Yaskawa INFORM job: BATMAN_4SPOINY2.JBI

/JOB
//NAME BATMAN_4SPOINY2
///FOLDERNAME KRIS-SCIANA
//POS
///NPOS 293,293,292,19,0,0
///TOOL 0
///POSTYPE PULSE
///PULSE
C00000=-27461,19727,-15013,-5964,93200,-7919
C00001=-53930,-34836,-43070,-10546,92631,44102
C00002=-59372,-32233,-36195,-10185,89087,42536
C00003=-59542,-32241,-35992,-10174,88938,42491
C00004=-59542,-32044,-34623,-10174,88208,42551
C00005=-59542,-32113,-35077,-10174,88448,42531
C00006=-60552,-31800,-34867,-10107,88354,42193
C00007=-59542,-32241,-35992,-10174,88938,42491
C00008=-64039,-48991,-58660,-9906,93649,40580
C00009=-69362,-49546,-56329,-9460,91325,38954
C00010=-72521,-45533,-52121,-9188,90441,37947
C00011=-72521,-45462,-50975,-9185,89780,37995
C00012=-72775,-45521,-51067,-9161,89777,37907
C00013=-73792,-45251,-50904,-9073,89701,37568
C00014=-72521,-45533,-52121,-9188,90441,37947
C00015=-72780,-67210,-74355,-9190,92926,37677
C00016=-104760,-79002,-75488,-1590,83769,-10908
C00017=-104760,-78316,-71792,-1595,81848,-10885
C00018=-104951,-72146,-66630,-1566,81838,-10949
C00019=-104951,-71873,-65349,-1567,81190,-10942
C00020=-104951,-71915,-65543,-1567,81288,-10943
C00021=-104860,-69153,-64201,-1578,81883,-10919
C00022=-104951,-72146,-66630,-1566,81838,-10949
C00023=-126930,-89810,-77004,2546,79326,-20912
C00024=-126930,-86182,-66696,2587,74851,-21005
C00025=-124517,-79688,-62407,2239,75475,-20152
C00026=-124517,-79051,-60693,2247,74749,-20166
C00027=-124517,-79260,-61250,2244,74984,-20162
C00028=-123686,-77088,-60280,2122,75480,-19864
C00029=-124517,-79688,-62407,2239,75475,-20152
C00030=-203387,-120314,-87249,1260,66339,-1853
C00031=-200667,-112422,-82916,708,67693,-857
C00032=-200667,-111236,-80756,708,66973,-859
C00033=-200667,-111296,-80865,708,67010,-859
C00034=-200121,-107908,-79763,595,68068,-656
C00035=-200667,-112422,-82916,708,67693,-857
C00036=-197903,-118206,-84689,161,65798,138
C00037=-190700,-136110,-79236,-12987,43309,5470
C00038=-193247,-133524,-78729,-11658,43940,4204
C00039=-193037,-133750,-78775,-11768,43882,4308
C00040=-191788,-131166,-76340,-12346,43888,4881
C00041=-190700,-136110,-79236,-12987,43309,5470
C00042=-159264,-85348,-72338,-26469,101848,35770
C00043=-164489,-85917,-58916,-26689,92487,35917
C00044=-168795,-82306,-57912,-27368,92208,34361
C00045=-170153,-80945,-57335,-27563,92069,33880
C00046=-170038,-81063,-57386,-27546,92081,33921
C00047=-169577,-79396,-55147,-27467,91768,34169
C00048=-168310,-82776,-58110,-27297,92259,34533
C00049=-174818,-166728,-104111,-5010,53468,9061
C00050=-151913,-165072,-108467,-9162,58894,17426
C00051=-31054,-58499,-67437,4813,86361,-7552
C00052=-17460,-13489,-32841,-5083,88285,10080
C00053=-18511,-10450,-28211,-4896,86939,9785
C00054=-18511,-10517,-26393,-4896,85789,9828
C00055=-18511,-10513,-26589,-4896,85911,9823
C00056=-19077,-8695,-25164,-4796,85935,9632
C00057=-18511,-10450,-28211,-4896,86939,9785
C00058=-19304,-17015,-37138,-4755,89006,9443
C00059=-40718,-16031,-27821,22618,89289,-5458
C00060=-35897,-12993,-23126,22071,86757,-4185
C00061=-35281,-10295,-21039,21995,86689,-3974
C00062=-35332,-10522,-21216,22001,86695,-3991
C00063=-35622,-10102,-19772,22045,86146,-4196
C00064=-35897,-12993,-23126,22071,86757,-4185
C00065=-31722,-22647,-27301,21597,83426,-3277
C00066=-29589,-18207,-23578,21312,82862,-2603
C00067=-29146,-15879,-21843,21245,82867,-2441
C00068=-29176,-16038,-21963,21249,82867,-2452
C00069=-29589,-15481,-20299,21334,82283,-2705
C00070=-29589,-18207,-23578,21312,82862,-2603
C00071=-33057,-35215,-50272,21725,90936,-2406
C00072=-13245,-10427,-29720,-5825,88219,11479
C00073=-13392,-4620,-21957,-5803,86422,11510
C00074=-18089,-7824,-24653,-4974,86126,9958
C00075=-18110,-8277,-24801,-4969,85982,9956
C00076=-21731,-10101,-26115,-4319,85651,8761
C00077=-21661,-10606,-26277,-4332,85495,8790
C00078=-25333,-12975,-27458,1213,84432,-1078
C00079=-19736,-16503,-27105,153,82354,789
C00080=-19363,-16615,-23205,6723,81452,-11372
C00081=-19940,-18075,-23614,6826,80998,-11595
C00082=-21964,-21673,-24603,7190,79942,-12350
C00083=-17410,-32379,-43825,-1943,88285,-427
C00084=-62758,-61083,-67514,-9356,96495,-3913
C00085=-199419,-126821,-93595,3849,72358,-1575
C00086=-214502,-101666,-82310,5387,79190,-6557
C00087=-215506,-95023,-76790,5488,79275,-6899
C00088=-206115,-95822,-76918,4502,78358,-3694
C00089=-205954,-96216,-76904,4488,78140,-3647
C00090=-199122,-96202,-76993,3725,77851,-1303
C00091=-199042,-96881,-76975,3719,77487,-1286
C00092=-188080,-119856,-79732,-8116,56883,3611
C00093=-198128,-125068,-78160,-5331,52444,-116
C00094=-199195,-125100,-74360,-11289,52271,7622
C00095=-182925,-108601,-69012,-21109,69501,28632
C00096=-173900,-101221,-64126,-22433,76310,30875
C00097=-171717,-100952,-63344,-22409,76572,31621
C00098=-165785,-126013,-84565,-21580,74443,34035
C00099=-65346,-79799,-84675,-10403,98195,30166
C00100=-73114,-35172,-46632,-9001,95792,24844
C00101=-73893,-33313,-43666,-8951,94846,24646
C00102=-56936,-3129,-12114,-26947,108321,27456
C00103=-55222,-19377,-25500,-26230,99599,30116
C00104=-48000,-22204,-22466,-25349,98847,33036
C00105=-47657,-23151,-32449,-25918,104076,32001
C00106=-58332,-49897,-67983,-12473,95404,30979
C00107=-76814,-87681,-77913,-12459,85852,4883
C00108=-98077,-64526,-65270,-10461,86864,-2540
C00109=-98077,-64172,-62734,-10473,85508,-2426
C00110=-98453,-62350,-60144,-10440,84814,-2496
C00111=-136928,-61997,-53571,24295,84631,-16368
C00112=-133428,-78274,-60683,19711,72960,-18904
C00113=-138454,-87211,-60543,20798,69473,-20912
C00114=-139028,-90281,-60991,20666,67739,-20449
C00115=-142002,-103150,-73880,19907,68072,-18980
C00116=-156669,-121711,-96887,11323,85539,-21769
C00117=-4467,-137969,-110669,6539,34039,3130
C00118=30106,49184,30056,7190,99242,80021
C00119=48667,-97469,-88024,4384,73291,-2494
C00120=49689,-78507,-72154,4117,73215,-2136
C00121=49303,-77230,-69865,4233,72483,-2298
C00122=49303,-77321,-70267,4229,72684,-2291
C00123=50594,-75678,-69509,3881,72996,-1827
C00124=50087,-79365,-72449,4017,72936,-2008
C00125=68843,-102719,-94603,-719,75306,4406
C00126=111940,-50312,-66287,845,90558,-21262
C00127=116747,-35795,-51410,28,88834,-19690
C00128=111075,-31135,-44901,14748,90637,-31106
C00129=112095,-31393,-44814,14616,90275,-30800
C00130=112020,-31375,-44802,14625,90290,-30824
C00131=111824,-29375,-42859,14647,90161,-30907
C00132=111075,-31135,-44901,14748,90637,-31106
C00133=115266,-12451,-41016,14369,96902,-28947
C00134=116842,-11754,-38964,14110,95764,-28553
C00135=117372,-11882,-38755,14027,95487,-28407
C00136=117096,-11854,-38735,14068,95534,-28493
C00137=116813,-10897,-37010,14093,95030,-28645
C00138=116549,-12463,-39204,14145,95601,-28669
C00139=116973,-27524,-54545,13255,91925,-29024
C00140=161629,-1767,-40127,-12706,111151,26907
C00141=160258,-5533,-27257,-16420,102000,26864
C00142=159800,-6307,-27168,-16383,101475,26773
C00143=160112,-5979,-26905,-16385,101541,26874
C00144=160141,-5574,-26041,-16363,101235,26926
C00145=160369,-6103,-29045,-16480,102795,26791
C00146=164567,12479,-21852,-12411,107740,28291
C00147=157312,-12873,-46942,3000,99665,-17174
C00148=206670,-20156,-47225,-4407,96533,-1302
C00149=207907,-5048,-28631,-4546,92932,-767
C00150=208193,-3786,-26509,-4582,92292,-649
C00151=208113,-4178,-26830,-4572,92282,-675
C00152=207509,-3531,-26303,-4488,92258,-873
C00153=208421,-5827,-28734,-4617,92624,-586
C00154=203791,-18365,-44572,-3987,95682,-2207
C00155=208102,-33244,-47535,-4348,72415,7516
C00156=208287,-28436,-43134,-4423,72190,7588
C00157=208434,-26310,-39925,-4502,71320,7672
C00158=208234,-36837,-41271,-4553,66735,7774
C00159=211009,-27621,-51707,-11614,93139,6311
C00160=152191,-52771,-83975,581,97487,43791
C00161=98829,-151569,-113617,-23423,60554,27083
C00162=63524,-95054,-80306,-9988,61383,12838
C00163=56536,-90563,-73566,-3171,58185,6546
C00164=56829,-88451,-72049,-3291,58345,6659
C00165=59876,-96663,-69219,-4945,52557,8119
C00166=60612,-96600,-68978,-5290,52489,8431
C00167=66960,-122601,-100767,717,65616,10335
C00168=151266,-17849,-52541,-13551,97671,36399
C00169=151622,-1723,-33362,-14991,96990,34005
C00170=151262,-1470,-31417,-14895,95899,34022
C00171=156478,-8848,-32076,-16260,93850,43651
C00172=161716,-19976,-35221,-16293,90376,44394
C00173=166380,-28542,-48041,-15538,92590,42053
C00174=176343,-26479,-59966,-14563,99290,38519
C00175=146432,-61605,-81283,-8581,90439,-5938
C00176=135076,-29257,-55178,-6049,90016,-9585
C00177=132700,-20433,-48103,-5503,90033,-10349
C00178=132491,-20005,-45954,-5452,88921,-10367
C00179=119630,-24773,-46451,11613,85271,-20135
C00180=112679,-48956,-51902,13552,77458,-23307
C00181=112569,-49156,-51831,13583,77335,-23359
C00182=106405,-53144,-61429,14838,82147,-24955
C00183=95224,-20248,-47255,12300,95289,-25611
C00184=95224,-20248,-47255,12300,95289,-25611
C00185=95567,-18089,-45671,12250,95373,-25491
C00186=-2669,-23033,-45877,12237,95351,-20479
C00187=-12882,-2605,-25335,12289,80797,-48712
C00188=-140228,6897,-12502,-16068,89102,25779
C00189=-178636,-27124,-21178,-9459,71149,14213
C00190=-190464,-2943,-638,1694,79970,9758
C00191=-190464,-2776,-23,1695,79677,9755
C00192=-190464,-2814,-164,1695,79744,9755
C00193=-190464,-1537,886,1697,79752,9755
C00194=-190079,-4348,-2686,1653,80502,9898
C00195=-170718,-9928,-4442,-11260,70728,17109
C00196=-176690,17572,15984,1100,84656,14555
C00197=-176690,17883,17124,1100,84116,14551
C00198=-176690,17847,16991,1100,84180,14551
C00199=-176937,19636,18668,1110,84073,14467
C00200=-176937,19636,18668,1110,84073,14467
C00201=-176690,17548,15886,1101,84706,14556
C00202=-159096,9684,11840,-13524,72569,21129
C00203=-163699,22746,22031,-3647,77400,19020
C00204=-163699,23053,23077,-3652,76914,19034
C00205=-163699,23004,22912,-3650,76991,19033
C00206=-164134,24645,24494,-3598,76842,18886
C00207=-163699,22706,21893,-3644,77465,19019
C00208=-150784,28408,29058,-15005,73089,24078
C00209=-157156,46221,45175,-1187,77129,21209
C00210=-157156,46539,46094,-1188,76728,21212
C00211=-157156,46464,45876,-1188,76822,21213
C00212=-157735,48153,47710,-1132,76554,21017
C00213=-157156,45966,44419,-1185,77462,21208
C00214=-142367,61055,63211,-16591,70629,27483
C00215=-154723,15756,14414,-2197,80088,22021
C00216=-154723,16062,15536,-2199,79553,22032
C00217=-154723,16000,15312,-2199,79658,22029
C00218=-155361,17628,16818,-2136,79550,21813
C00219=-154295,14517,12085,-2236,80891,22153
C00220=-151769,-34490,-30946,-14563,77368,23201
C00221=-173063,-38776,-28238,-10774,70233,16311
C00222=-172381,-31676,-18222,-12843,69119,19791
C00223=-189396,-43787,-25561,-9322,65102,13897
C00224=-212287,-48657,-28204,-3544,62394,5501
C00225=-221997,-47169,-27328,-892,62356,1858
C00226=-221072,-57002,-35060,1210,62084,-1011
C00227=-183831,-45924,-33017,621,66496,-211
C00228=-184325,-38707,-22706,764,63866,-409
C00229=-169590,-26315,-14874,-3175,65639,5020
C00230=-153390,-792,4257,-7245,68027,10841
C00231=-148403,11895,15303,-8450,68237,12643
C00232=-147332,15315,18416,-8713,68194,13036
C00233=-141966,-23744,-26450,-9578,76254,14345
C00234=-49773,-23801,-26487,-9571,76243,10777
C00235=-11499,-92934,-63711,-14704,67160,23123
C00236=5078,129767,24381,-2980,99042,84457
C00237=-23281,115763,31203,9131,91877,90037
C00238=-55336,37368,-13455,9130,92546,90074
C00239=-110497,-96700,-87975,9097,92672,90031
C00240=-122519,-98627,-88731,8985,93501,45120
C00241=-122519,-98627,-88731,8985,93501,45120
C00242=-231043,-103510,-90228,-14600,66848,14562
C00243=-239015,-52899,-63453,-12354,87389,13057
C00244=-232211,-37055,-48018,-13457,87263,15389
C00245=-232200,-37444,-47619,-13460,86829,15441
C00246=-232200,-37417,-46208,-13467,85999,15531
C00247=-232200,-37422,-46357,-13466,86086,15522
C00248=-232546,-36405,-45702,-13410,86146,15397
C00249=-232526,-38013,-47982,-13409,86709,15341
C00250=-213204,-18706,-38315,-16054,93998,21087
C00251=-215284,-13076,-30615,-15755,91824,20653
C00252=-215284,-13133,-29398,-15744,91072,20748
C00253=-215284,-13128,-29540,-15745,91159,20737
C00254=-215902,-11928,-28618,-15673,91088,20532
C00255=-215392,-13382,-30849,-15743,91789,20621
C00256=-206438,9841,-12512,-16716,94160,23395
C00257=-205120,11503,-10315,-16825,93948,23882
C00258=-205120,11440,-9133,-16804,93220,23984
C00259=-205120,11443,-9214,-16804,93269,23978
C00260=-205697,12454,-8305,-16750,93115,23798
C00261=-205222,11014,-10755,-16815,93943,23847
C00262=-210286,16144,-6103,-16310,92719,22261
C00263=-208996,19538,-3176,-16442,92919,22681
C00264=-208996,19485,-1978,-16424,92184,22779
C00265=-208996,19488,-2094,-16426,92254,22769
C00266=-209668,20896,-770,-16357,92032,22565
C00267=-208996,19564,-3616,-16449,93191,22643
C00268=-202176,43267,18401,-17042,93256,25006
C00269=-201249,45778,22861,-17085,92051,25496
C00270=-201249,45831,24224,-17069,91274,25603
C00271=-201249,45825,24100,-17070,91344,25593
C00272=-201817,46846,25195,-17022,91083,25430
C00273=-201596,44518,21658,-17057,92067,25371
C00274=-210187,6216,-22915,-16512,97781,21615
C00275=-216436,-2522,-24538,-15653,93231,20080
C00276=-219720,2451,-17856,-13270,92091,26137
C00277=-232169,-16488,-32780,-11683,89671,22159
C00278=-226973,-31382,-43065,-12371,89135,23971
C00279=-237194,-42183,-49809,-10971,86308,20756
C00280=-231421,-47421,-61288,-11801,91394,22246
C00281=-231421,-47421,-61288,-11801,91394,22246
C00282=-240248,-57151,-63303,-3936,83174,7432
C00283=-224450,-39830,-53255,-6930,86930,12556
C00284=-211441,-17782,-38439,-9211,90387,16662
C00285=-206434,-6086,-29592,-10033,91526,18242
C00286=-205798,-3820,-27691,-10133,91599,18448
C00287=-200228,-22351,-51424,-11111,97297,19798
C00288=-129551,-116321,-98683,-1361,90461,40912
C00289=-129551,-116321,-98683,-1361,90461,40912
C00290=-59952,-112124,-97380,-1385,91667,40557
C00291=-59953,-112125,-97379,-1385,91667,40556
C00292=1527,-36481,-34263,-1012,58134,86073
BC00000=81460,853554,487182
BC00001=164754,872951,482279
BC00002=164754,872951,482279
BC00003=164754,872951,482279
BC00004=164754,872951,482279
BC00005=164754,872951,482279
BC00006=164754,872951,482279
BC00007=164754,872951,482279
BC00008=164754,872951,482279
BC00009=164754,872951,482279
BC00010=164754,872951,482279
BC00011=164754,872951,482279
BC00012=164754,872951,482279
BC00013=164754,872951,482279
BC00014=164754,872951,482279
BC00015=164754,872951,482279
BC00016=164754,872951,482279
BC00017=164754,872951,482279
BC00018=164754,872951,482279
BC00019=164754,872951,482279
BC00020=164754,872951,482279
BC00021=164754,872951,482279
BC00022=164754,872951,482279
BC00023=164754,872951,482279
BC00024=164754,872951,482279
BC00025=164754,872951,482279
BC00026=164754,872951,482279
BC00027=164754,872951,482279
BC00028=164754,872951,482279
BC00029=164754,872951,482279
BC00030=164754,872951,482279
BC00031=164754,872951,482279
BC00032=164754,872951,482279
BC00033=164754,872951,482279
BC00034=164754,872951,482279
BC00035=164754,872951,482279
BC00036=164754,872951,482279
BC00037=164754,872951,482279
BC00038=164754,872951,482279
BC00039=164754,872951,482279
BC00040=164754,872951,482279
BC00041=164754,872951,482279
BC00042=164753,872951,482277
BC00043=164753,872950,482272
BC00044=164753,872950,482272
BC00045=164753,872950,482272
BC00046=164753,872950,482272
BC00047=164753,872950,482272
BC00048=164753,872950,482272
BC00049=164754,872951,482279
BC00050=164754,872951,482279
BC00051=164754,872951,482279
BC00052=164754,872951,482279
BC00053=164754,872951,482279
BC00054=164754,872951,482279
BC00055=164754,872951,482279
BC00056=164754,872951,482279
BC00057=164754,872951,482279
BC00058=164754,872951,482279
BC00059=164754,872951,482279
BC00060=164754,872951,482279
BC00061=164754,872951,482279
BC00062=164754,872951,482279
BC00063=164754,872951,482279
BC00064=164754,872951,482279
BC00065=164754,872951,482279
BC00066=164754,872951,482279
BC00067=164754,872951,482279
BC00068=164754,872951,482279
BC00069=164754,872951,482279
BC00070=164754,872951,482279
BC00071=164754,872951,482279
BC00072=164754,872951,482279
BC00073=164754,872951,482279
BC00074=164754,872951,482279
BC00075=164754,872951,482279
BC00076=164754,872951,482279
BC00077=164754,872951,482279
BC00078=164754,872951,482279
BC00079=164754,872951,482279
BC00080=164754,872951,482279
BC00081=164754,872951,482279
BC00082=164754,872951,482279
BC00083=164755,872951,482282
BC00084=164755,872950,618004
BC00085=164755,872950,482279
BC00086=164755,872950,482279
BC00087=164755,872950,482279
BC00088=164755,872950,482279
BC00089=164755,872950,482279
BC00090=164755,872950,482279
BC00091=164755,872950,482279
BC00092=164755,872950,482279
BC00093=164755,872950,482279
BC00094=164755,872950,482279
BC00095=164755,872950,482279
BC00096=164755,872950,482279
BC00097=164755,872950,482279
BC00098=164755,872950,482279
BC00099=164755,872950,482279
BC00100=164755,872950,482279
BC00101=164755,872950,482279
BC00102=164755,872950,482279
BC00103=164755,872950,482279
BC00104=164755,872950,482279
BC00105=164755,872950,482279
BC00106=164755,872950,482279
BC00107=164755,872950,482279
BC00108=164755,872950,482279
BC00109=164755,872950,482279
BC00110=164755,872950,482279
BC00111=164755,872950,482279
BC00112=164755,872950,482279
BC00113=164755,872950,482279
BC00114=164755,872950,482279
BC00115=164755,872950,482279
BC00116=164755,872950,715358
BC00117=113180,1185778,1059182
BC00118=126121,1185200,1068204
BC00119=256124,1186110,610519
BC00120=256124,1186110,610519
BC00121=256124,1186110,610519
BC00122=256124,1186110,610519
BC00123=256124,1186110,610519
BC00124=256124,1186110,610519
BC00125=256124,1186110,610519
BC00126=256124,1186110,610519
BC00127=256124,1186110,610519
BC00128=256124,1186110,610519
BC00129=256124,1186110,610519
BC00130=256124,1186110,610519
BC00131=256124,1186110,610519
BC00132=256124,1186110,610519
BC00133=256124,1186110,610519
BC00134=256124,1186110,610519
BC00135=256124,1186110,610519
BC00136=256124,1186110,610519
BC00137=256124,1186110,610519
BC00138=256124,1186110,610519
BC00139=256124,1186110,610519
BC00140=256124,1186110,610519
BC00141=256124,1186110,610519
BC00142=256124,1186110,610519
BC00143=256124,1186110,610519
BC00144=256124,1186110,610519
BC00145=256124,1186110,610519
BC00146=256124,1186110,610519
BC00147=256124,1186110,610519
BC00148=256124,1186110,610519
BC00149=256124,1186110,610519
BC00150=256124,1186110,610519
BC00151=256124,1186110,610519
BC00152=256124,1186110,610519
BC00153=256124,1186110,610519
BC00154=256124,1186110,610519
BC00155=256124,1186110,610519
BC00156=256124,1186110,610519
BC00157=256124,1186110,610519
BC00158=256124,1186110,610519
BC00159=256124,1186110,610519
BC00160=256123,1186110,610516
BC00161=256123,1186110,610516
BC00162=256123,1186110,610516
BC00163=256123,1186110,610516
BC00164=256122,1186109,610509
BC00165=256122,1186109,610509
BC00166=256122,1186109,610509
BC00167=256122,1186109,610509
BC00168=256122,1186109,610509
BC00169=256122,1186109,610507
BC00170=256122,1186109,610507
BC00171=256122,1186109,610507
BC00172=256122,1186109,610507
BC00173=256122,1186109,610507
BC00174=256122,1186109,610507
BC00175=256122,1186109,610507
BC00176=256123,1186109,610505
BC00177=256123,1186109,610505
BC00178=256123,1186109,610505
BC00179=256123,1186109,610505
BC00180=256123,1186109,610505
BC00181=256123,1186109,610505
BC00182=256123,1186109,610505
BC00183=256123,1186109,1047068
BC00184=365218,1186109,1047068
BC00185=346946,697413,1047068
BC00186=120788,697413,1047068
BC00187=122987,697175,1055782
BC00188=316946,696835,347311
BC00189=316946,814999,347311
BC00190=316946,814999,347311
BC00191=316946,814999,347311
BC00192=316946,814999,347311
BC00193=316946,814999,347311
BC00194=316946,814999,347311
BC00195=316946,814999,347311
BC00196=316946,814999,347311
BC00197=316946,814999,347311
BC00198=316946,814999,347311
BC00199=316946,814999,347311
BC00200=316946,814999,347311
BC00201=316946,814999,347311
BC00202=316946,814999,347311
BC00203=316946,814999,347311
BC00204=316946,814999,347311
BC00205=316946,814999,347311
BC00206=316946,814999,347311
BC00207=316946,814999,347311
BC00208=316946,814999,347311
BC00209=316946,814999,347311
BC00210=316946,814999,347311
BC00211=316946,814999,347311
BC00212=316946,814999,347311
BC00213=316946,814999,347311
BC00214=316946,814999,347311
BC00215=316946,880782,347311
BC00216=316946,880782,347311
BC00217=316946,880782,347311
BC00218=316946,880782,347311
BC00219=316946,880782,347311
BC00220=316946,880782,347311
BC00221=316946,880782,347311
BC00222=316944,880782,347309
BC00223=316944,880782,347309
BC00224=316944,880782,347309
BC00225=316944,880782,347309
BC00226=316944,880782,347309
BC00227=316944,880782,347309
BC00228=316944,880782,347309
BC00229=316944,880782,347309
BC00230=316944,880782,347309
BC00231=316944,880782,347309
BC00232=316944,880782,347309
BC00233=316944,880783,347308
BC00234=222554,686457,538102
BC00235=140072,681044,975858
BC00236=125092,679971,1067929
BC00237=86290,680534,1057546
BC00238=245616,676469,1003930
BC00239=394456,788206,911844
BC00240=397244,925267,911844
BC00241=397244,1175961,911844
BC00242=390474,1092114,192725
BC00243=395058,1054624,192725
BC00244=395058,1054624,192721
BC00245=395058,1054624,192721
BC00246=395058,1054624,192721
BC00247=395058,1054624,192721
BC00248=395058,1054624,192721
BC00249=395058,1054624,192721
BC00250=395058,1054624,192721
BC00251=395058,1054625,192719
BC00252=395058,1054625,192719
BC00253=395058,1054625,192719
BC00254=395058,1054625,192719
BC00255=395058,1054625,192719
BC00256=395058,1054625,192719
BC00257=395058,1054625,192719
BC00258=395058,1054625,192719
BC00259=395058,1054625,192719
BC00260=395058,1054625,192719
BC00261=395058,1054625,192719
BC00262=395058,1091493,192719
BC00263=395058,1091493,192719
BC00264=395058,1091493,192719
BC00265=395058,1091493,192719
BC00266=395058,1091493,192719
BC00267=395058,1091493,192719
BC00268=395058,1091493,192719
BC00269=395058,1091493,192719
BC00270=395058,1091493,192719
BC00271=395058,1091493,192719
BC00272=395058,1091493,192719
BC00273=395058,1091493,192719
BC00274=395058,1091493,192719
BC00275=395058,1091493,192719
BC00276=395058,1091493,192719
BC00277=395058,1091493,192719
BC00278=395058,1041797,192719
BC00279=395058,1041797,192719
BC00280=395058,1041797,192719
BC00281=348075,1128251,164723
BC00282=348075,1128251,164723
BC00283=348075,1128251,164723
BC00284=348075,1128251,164723
BC00285=348075,1128251,164723
BC00286=348075,1128251,164723
BC00287=348075,1146299,164723
BC00288=396108,1148564,1054955
BC00289=396108,821890,1054955
BC00290=393986,698880,773470
BC00291=393986,698880,773468
BC00292=65416,672013,1068190
EC00000=811452,1111165
EC00001=811450,1111165
EC00002=811450,1111165
EC00003=811450,1111165
EC00004=811450,1111165
EC00005=811450,1111165
EC00006=811450,1111165
EC00007=811450,1111165
EC00008=811450,1111165
EC00009=811450,1111165
EC00010=811450,1111165
EC00011=811450,1111165
EC00012=811450,1111165
EC00013=811450,1111165
EC00014=811450,1111165
EC00015=811450,1111165
EC00016=811450,1111165
EC00017=811450,1111165
EC00018=811450,1111165
EC00019=811450,1111165
EC00020=811450,1111165
EC00021=811450,1111165
EC00022=811450,1111165
EC00023=811450,1111165
EC00024=811450,1111165
EC00025=811450,1111165
EC00026=811450,1111165
EC00027=811450,1111165
EC00028=811450,1111165
EC00029=811450,1111165
EC00030=811450,1111165
EC00031=811450,1111165
EC00032=811450,1111165
EC00033=811450,1111165
EC00034=811450,1111165
EC00035=811450,1111165
EC00036=811450,1111165
EC00037=811450,1111165
EC00038=811450,1111165
EC00039=811450,1111165
EC00040=811450,1111165
EC00041=811450,1111165
EC00042=811447,1111166
EC00043=811443,1111166
EC00044=811443,1111166
EC00045=811443,1111166
EC00046=811443,1111166
EC00047=811443,1111166
EC00048=811443,1111166
EC00049=811450,1111165
EC00050=811450,1111165
EC00051=811450,1111165
EC00052=811450,1111165
EC00053=811450,1111165
EC00054=811450,1111165
EC00055=811450,1111165
EC00056=811450,1111165
EC00057=811450,1111165
EC00058=811450,1111165
EC00059=811450,1111165
EC00060=811450,1111165
EC00061=811450,1111165
EC00062=811450,1111165
EC00063=811450,1111165
EC00064=811450,1111165
EC00065=811450,1111165
EC00066=811450,1111165
EC00067=811450,1111165
EC00068=811450,1111165
EC00069=811450,1111165
EC00070=811450,1111165
EC00071=811450,1111165
EC00072=811450,1111165
EC00073=811450,1111165
EC00074=811450,1111165
EC00075=811450,1111165
EC00076=811450,1111165
EC00077=811450,1111165
EC00078=811450,1111165
EC00079=811450,1111165
EC00080=811450,1111165
EC00081=811450,1111165
EC00082=811450,1111165
EC00083=811452,1111165
EC00084=811451,1111165
EC00085=811451,1111165
EC00086=811451,1111165
EC00087=811451,1111165
EC00088=811451,1111165
EC00089=811451,1111165
EC00090=811451,1111165
EC00091=811451,1111165
EC00092=811451,1111165
EC00093=811451,1111165
EC00094=811451,1111165
EC00095=811451,1111165
EC00096=811451,1111165
EC00097=811451,1111165
EC00098=811451,1111165
EC00099=811451,1111165
EC00100=811451,1111165
EC00101=811451,1111165
EC00102=811451,1111165
EC00103=811451,1111165
EC00104=811451,1111165
EC00105=811451,1111165
EC00106=811451,1111165
EC00107=811451,1111165
EC00108=811451,1111165
EC00109=811451,1111165
EC00110=811451,1111165
EC00111=811451,1111165
EC00112=811451,1111165
EC00113=811451,1111165
EC00114=811451,1111165
EC00115=811451,1111165
EC00116=811451,1111165
EC00117=363208,1107222
EC00118=363208,1107222
EC00119=363208,1107222
EC00120=363208,1107222
EC00121=363208,1107222
EC00122=363208,1107222
EC00123=363208,1107222
EC00124=363208,1107222
EC00125=363208,1107222
EC00126=363208,1107222
EC00127=363208,1107222
EC00128=363208,1107222
EC00129=363208,1107222
EC00130=363208,1107222
EC00131=363208,1107222
EC00132=363208,1107222
EC00133=363208,1107222
EC00134=363208,1107222
EC00135=363208,1107222
EC00136=363208,1107222
EC00137=363208,1107222
EC00138=363208,1107222
EC00139=363208,1107222
EC00140=363208,1107222
EC00141=363208,1107222
EC00142=363208,1107222
EC00143=363208,1107222
EC00144=363208,1107222
EC00145=363208,1107222
EC00146=363208,1107222
EC00147=363208,1107222
EC00148=363208,1107222
EC00149=363208,1107222
EC00150=363208,1107222
EC00151=363208,1107222
EC00152=363208,1107222
EC00153=363208,1107222
EC00154=363208,1107222
EC00155=363208,1107222
EC00156=363208,1107222
EC00157=363208,1107222
EC00158=363208,1107222
EC00159=363208,1107222
EC00160=363208,1107222
EC00161=363208,1107222
EC00162=363208,1107222
EC00163=363208,1107222
EC00164=363207,1107222
EC00165=363207,1107222
EC00166=363207,1107222
EC00167=363207,1107222
EC00168=363207,1107222
EC00169=363206,1107222
EC00170=363206,1107222
EC00171=363206,1107222
EC00172=363206,1107222
EC00173=363206,1107222
EC00174=363206,1107222
EC00175=363206,1107222
EC00176=363206,1107222
EC00177=363206,1107222
EC00178=363206,1107222
EC00179=363206,1107222
EC00180=363206,1107222
EC00181=363206,1107222
EC00182=363206,1107222
EC00183=363206,1107222
EC00184=363206,1107222
EC00185=0,556476
EC00186=802750,556476
EC00187=802750,556476
EC00188=802750,556476
EC00189=802750,556476
EC00190=802750,556476
EC00191=802750,556476
EC00192=802750,556476
EC00193=802750,556476
EC00194=802750,556476
EC00195=802750,556476
EC00196=802750,556476
EC00197=802750,556476
EC00198=802750,556476
EC00199=802750,556476
EC00200=802750,556476
EC00201=802750,556476
EC00202=802750,556476
EC00203=802750,556476
EC00204=802750,556476
EC00205=802750,556476
EC00206=802750,556476
EC00207=802750,556476
EC00208=802750,556476
EC00209=802750,556476
EC00210=802750,556476
EC00211=802750,556476
EC00212=802750,556476
EC00213=802750,556476
EC00214=802750,556476
EC00215=802750,556476
EC00216=802750,556476
EC00217=802750,556476
EC00218=802750,556476
EC00219=802750,556476
EC00220=802750,556476
EC00221=802749,556476
EC00222=802749,556476
EC00223=802749,556476
EC00224=802749,556476
EC00225=802749,556476
EC00226=802749,556476
EC00227=802749,556476
EC00228=802749,556476
EC00229=802749,556476
EC00230=802749,556476
EC00231=802749,556476
EC00232=802748,556476
EC00233=802748,556476
EC00234=-793507,556476
EC00235=-793506,556477
EC00236=-793506,556477
EC00237=-793506,556477
EC00238=-793506,556477
EC00239=-793506,556477
EC00240=-793506,556477
EC00241=-793506,556477
EC00242=-793506,556477
EC00243=-793505,556477
EC00244=-793505,556477
EC00245=-793505,556477
EC00246=-793505,556477
EC00247=-793505,556477
EC00248=-793505,556477
EC00249=-793505,556477
EC00250=-793504,556477
EC00251=-793504,556477
EC00252=-793504,556477
EC00253=-793504,556477
EC00254=-793504,556477
EC00255=-793504,556477
EC00256=-793504,556477
EC00257=-793504,556477
EC00258=-793504,556477
EC00259=-793504,556477
EC00260=-793504,556477
EC00261=-793504,556477
EC00262=-793504,556477
EC00263=-793504,556477
EC00264=-793504,556477
EC00265=-793504,556477
EC00266=-793504,556477
EC00267=-793504,556477
EC00268=-793504,556477
EC00269=-793504,556477
EC00270=-793504,556477
EC00271=-793504,556477
EC00272=-793504,556477
EC00273=-793504,556477
EC00274=-793504,556477
EC00275=-793504,556477
EC00276=-793504,556477
EC00277=-793504,556477
EC00278=-793504,556477
EC00279=-793504,556477
EC00280=-793504,556477
EC00281=-793504,556477
EC00282=-793504,556477
EC00283=-793504,556477
EC00284=-793504,556477
EC00285=-793504,556477
EC00286=-793504,556477
EC00287=-793504,556477
EC00288=-793504,556477
EC00289=-793504,556477
EC00290=-793503,8052
EC00291=0,556477
///POSTYPE BASE
///RECTAN
///RCONF 0,0,0,0,0,0,0,0,0,0,0,0,0,0,0,0,0,0,0,0,0,0,0,0
P00006=0.000,0.000,0.000,0.0000,0.0000,0.0000
P00021=-0.339,1.359,3.368,0.0000,0.0000,0.0000
P00022=-0.114,-0.780,3.887,0.0000,0.0000,0.0000
P00023=0.143,-0.036,0.682,0.0000,0.0000,0.0000
P00024=0.011,-0.011,1.365,0.0000,0.0000,0.0000
P00025=2.242,-0.049,-1.961,0.0000,0.0000,0.0000
P00026=0.572,-0.002,0.234,0.0000,0.0000,0.0000
P00027=-0.746,0.015,-9.096,0.0000,0.0000,0.0000
P00028=-2.237,-0.018,-7.702,0.0000,0.0000,0.0000
P00029=-2.156,-0.086,-4.681,0.0000,0.0000,0.0000
P00030=5.926,-4.294,-1.390,0.0000,0.0000,0.0000
P00034=-0.304,0.773,-2.693,0.0000,0.0000,0.0000
P00035=2.817,0.591,-1.622,0.0000,0.0000,0.0000
P00036=-1.108,-0.829,1.850,0.0000,0.0000,0.0000
P00037=0.023,0.937,-2.677,0.0000,0.0000,0.0000
P00040=-0.030,9.648,2.467,0.0000,0.0000,0.0000
P00041=0.192,3.924,0.305,0.0000,0.0000,0.0000
P00042=-0.217,1.941,0.413,0.0000,0.0000,0.0000
P00043=-0.044,-1.937,1.197,0.0000,0.0000,0.0000
//INST
///DATE 2024/07/30 22:39
///ATTR SC,RW
///GROUP1 RB1,BS1
///GROUP2 ST1
NOP
SFTOF3D
SFTOF
SSFTOF
MOVJ C00000 BC00000 VJ=100.00  +MOVJ EC00000 VJ=100.00
'SZUKANIE
SFTOF3D
MOVJ C00001 BC00001 VJ=100.00  +MOVJ EC00001 VJ=30.00
MOVL C00002 BC00002 V=83.3  +MOVJ EC00002 VJ=15.00
MOVL C00003 BC00003 V=83.3  +MOVJ EC00003 VJ=15.00
SREFP 3 C00004 BC00004  +REFP EC00004
CALL JOB:SEARCH-R1-S13D
SET P026 P006
SFTON3D P026
MOVL C00005 BC00005 V=83.3  +MOVJ EC00005 VJ=15.00
SREFP 3 C00006 BC00006  +REFP EC00006
CALL JOB:SEARCH-R1-S13D
SET P026 P006
MOVL C00007 BC00007 V=83.3  +MOVJ EC00007 VJ=15.00
SFTOF3D
MOVL C00008 BC00008 V=83.3  +MOVJ EC00008 VJ=15.00
MOVL C00009 BC00009 V=83.3  +MOVJ EC00009 VJ=15.00
MOVL C00010 BC00010 V=83.3  +MOVJ EC00010 VJ=15.00
SREFP 3 C00011 BC00011  +REFP EC00011
CALL JOB:SEARCH-R1-S13D
SET P027 P006
SFTON3D P027
MOVL C00012 BC00012 V=83.3  +MOVJ EC00012 VJ=15.00
SREFP 3 C00013 BC00013  +REFP EC00013
CALL JOB:SEARCH-R1-S13D
SET P027 P006
MOVL C00014 BC00014 V=83.3  +MOVJ EC00014 VJ=15.00
SFTOF3D
MOVJ C00015 BC00015 VJ=100.00  +MOVJ EC00015 VJ=100.00
SFTOF3D
MOVJ C00016 BC00016 VJ=100.00  +MOVJ EC00016 VJ=100.00
MOVL C00017 BC00017 V=83.3  +MOVJ EC00017 VJ=15.00
MOVL C00018 BC00018 V=83.3  +MOVJ EC00018 VJ=15.00
SREFP 3 C00019 BC00019  +REFP EC00019
CALL JOB:SEARCH-R1-S13D
SET P029 P006
SFTON3D P029
MOVL C00020 BC00020 V=83.3  +MOVJ EC00020 VJ=15.00
SREFP 3 C00021 BC00021  +REFP EC00021
CALL JOB:SEARCH-R1-S13D
SET P029 P006
MOVL C00022 BC00022 V=83.3  +MOVJ EC00022 VJ=15.00
SFTOF3D
MOVL C00023 BC00023 V=83.3  +MOVJ EC00023 VJ=15.00
MOVL C00024 BC00024 V=83.3  +MOVJ EC00024 VJ=15.00
MOVL C00025 BC00025 V=83.3  +MOVJ EC00025 VJ=15.00
SREFP 3 C00026 BC00026  +REFP EC00026
CALL JOB:SEARCH-R1-S13D
SET P030 P006
SFTON3D P030
MOVL C00027 BC00027 V=83.3  +MOVJ EC00027 VJ=15.00
SREFP 3 C00028 BC00028  +REFP EC00028
CALL JOB:SEARCH-R1-S13D
SET P030 P006
MOVL C00029 BC00029 V=83.3  +MOVJ EC00029 VJ=15.00
SFTOF3D
MOVL C00030 BC00030 V=250.0  +MOVJ EC00030 VJ=15.00
MOVL C00031 BC00031 V=83.3  +MOVJ EC00031 VJ=15.00
SREFP 3 C00032 BC00032  +REFP EC00032
CALL JOB:SEARCH-R1-S13D
SET P036 P006
SFTON3D P036
MOVL C00033 BC00033 V=83.3  +MOVJ EC00033 VJ=15.00
SREFP 3 C00034 BC00034  +REFP EC00034
CALL JOB:SEARCH-R1-S13D
SET P036 P006
MOVL C00035 BC00035 V=83.3  +MOVJ EC00035 VJ=15.00
SFTOF3D
MOVL C00036 BC00036 V=333.3  +MOVJ EC00036 VJ=0.78
MOVL C00037 BC00037 V=200.0  +MOVJ EC00037 VJ=15.00
SREFP 3 C00038 BC00038  +REFP EC00038
CALL JOB:SEARCH-R1-S13D
SET P040 P006
SFTON3D P040
MOVL C00039 BC00039 V=83.3  +MOVJ EC00039 VJ=15.00
SREFP 3 C00040 BC00040  +REFP EC00040
CALL JOB:SEARCH-R1-S13D
SET P040 P006
MOVL C00041 BC00041 V=83.3  +MOVJ EC00041 VJ=15.00
SFTOF3D
MOVJ C00042 BC00042 VJ=100.00  +MOVJ EC00042 VJ=0.78
MOVJ C00043 BC00043 VJ=100.00  +MOVJ EC00043 VJ=100.00
MOVL C00044 BC00044 V=166.7  +MOVJ EC00044 VJ=15.00
SREFP 3 C00045 BC00045  +REFP EC00045
CALL JOB:SEARCH-R1-S13D
SET P041 P006
SFTON3D P041
MOVL C00046 BC00046 V=83.3  +MOVJ EC00046 VJ=15.00
SREFP 3 C00047 BC00047  +REFP EC00047
CALL JOB:SEARCH-R1-S13D
SET P041 P006
MOVL C00048 BC00048 V=83.3  +MOVJ EC00048 VJ=15.00
SFTOF3D
MOVL C00049 BC00049 V=250.0  +MOVJ EC00049 VJ=15.00
MOVJ C00050 BC00050 VJ=100.00  +MOVJ EC00050 VJ=15.00
MOVJ C00051 BC00051 VJ=100.00  +MOVJ EC00051 VJ=100.00
MOVJ C00052 BC00052 VJ=100.00  +MOVJ EC00052 VJ=100.00
MOVL C00053 BC00053 V=166.7  +MOVJ EC00053 VJ=15.00
SREFP 3 C00054 BC00054  +REFP EC00054
CALL JOB:SEARCH-R1-S13D
SET P037 P006
SFTON3D P037
MOVL C00055 BC00055 V=83.3  +MOVJ EC00055 VJ=15.00
SREFP 3 C00056 BC00056  +REFP EC00056
CALL JOB:SEARCH-R1-S13D
SET P037 P006
MOVL C00057 BC00057 V=83.3  +MOVJ EC00057 VJ=15.00
SFTOF3D
MOVJ C00058 BC00058 VJ=100.00  +MOVJ EC00058 VJ=100.00
MOVJ C00059 BC00059 VJ=100.00  +MOVJ EC00059 VJ=100.00
MOVL C00060 BC00060 V=83.3  +MOVJ EC00060 VJ=15.00
SREFP 3 C00061 BC00061  +REFP EC00061
CALL JOB:SEARCH-R1-S13D
SET P042 P006
SFTOF3D
SFTON3D P042
MOVL C00062 BC00062 V=83.3  +MOVJ EC00062 VJ=15.00
SREFP 3 C00063 BC00063  +REFP EC00063
CALL JOB:SEARCH-R1-S13D
SET P042 P006
MOVL C00064 BC00064 V=83.3  +MOVJ EC00064 VJ=15.00
SFTOF3D
MOVJ C00065 BC00065 VJ=100.00  +MOVJ EC00065 VJ=100.00
MOVL C00066 BC00066 V=166.7  +MOVJ EC00066 VJ=15.00
SREFP 3 C00067 BC00067  +REFP EC00067
CALL JOB:SEARCH-R1-S13D
SET P042 P006
SFTON3D P042
MOVL C00068 BC00068 V=83.3  +MOVJ EC00068 VJ=15.00
SREFP 3 C00069 BC00069  +REFP EC00069
CALL JOB:SEARCH-R1-S13D
SET P042 P006
MOVL C00070 BC00070 V=83.3  +MOVJ EC00070 VJ=15.00
SFTOF3D
MOVJ C00071 BC00071 VJ=100.00  +MOVJ EC00071 VJ=100.00
SFTOF3D
MOVL C00072 BC00072 V=166.7  +MOVJ EC00072 VJ=15.00
SFTON3D P037
MACRO1 MJ#(0) ARGF7
SMOVL C00073 BC00073 V=166.7  +MOVJ EC00073
ARCON
SMOVL C00074 BC00074 V=10.0  +MOVJ EC00074
SMOVL C00075 BC00075 V=10.0  +MOVJ EC00075
SMOVL C00076 BC00076 V=10.0  +MOVJ EC00076
SMOVL C00077 BC00077 V=10.0  +MOVJ EC00077
SMOVL C00078 BC00078 V=10.0  +MOVJ EC00078
SFTOF3D
SFTON3D P042
SMOVL C00079 BC00079 V=10.0  +MOVJ EC00079
SFTOF3D
SFTON3D P043
SMOVL C00080 BC00080 V=10.0  +MOVJ EC00080
MACRO1 MJ#(0) ARGF7
SMOVL C00081 BC00081 V=10.0  +MOVJ EC00081
SMOVL C00082 BC00082 V=10.0  +MOVJ EC00082
ARCOF
MOVJ C00083 BC00083 VJ=20.00  +MOVJ EC00083 VJ=20.00
SFTOF3D
MOVJ C00084 BC00084 VJ=100.00  +MOVJ EC00084 VJ=20.00
MOVJ C00085 BC00085 VJ=100.00  +MOVJ EC00085 VJ=20.00
SFTON3D P036
MOVJ C00086 BC00086 VJ=20.00  +MOVJ EC00086 VJ=100.00
SMOVL C00087 BC00087 V=250.0  +MOVJ EC00087
ARCON
SMOVL C00088 BC00088 V=10.0  +MOVJ EC00088
TIMER T=0.10
SMOVL C00089 BC00089 V=10.0  +MOVJ EC00089
SMOVL C00090 BC00090 V=10.0  +MOVJ EC00090
SMOVL C00091 BC00091 V=10.0  +MOVJ EC00091
SMOVL C00092 BC00092 V=10.0  +MOVJ EC00092
SFTOF3D
SFTON3D P040
SMOVL C00093 BC00093 V=10.0  +MOVJ EC00093
SMOVL C00094 BC00094 V=10.0  +MOVJ EC00094
SFTOF3D
SFTON3D P041
SMOVL C00095 BC00095 V=10.0  +MOVJ EC00095
ARCON
SMOVL C00096 BC00096 V=10.0  +MOVJ EC00096
SMOVL C00097 BC00097 V=10.0  +MOVJ EC00097
ARCOF
MOVJ C00098 BC00098 VJ=15.00  +MOVJ EC00098 VJ=15.00
SFTOF3D
MOVJ C00099 BC00099 VJ=30.00  +MOVJ EC00099 VJ=30.00
SFTON3D P027
MOVJ C00100 BC00100 VJ=30.00  +MOVJ EC00100 VJ=30.00
SMOVL C00101 BC00101 V=250.0  +MOVJ EC00101
ARCON
SMOVL C00102 BC00102 V=10.0  +MOVJ EC00102
SFTOF3D
SFTON3D P026
SMOVL C00103 BC00103 V=10.0  +MOVJ EC00103
SMOVL C00104 BC00104 V=10.0  +MOVJ EC00104
ARCOF
SFTOF3D
MOVJ C00105 BC00105 VJ=100.00  +MOVJ EC00105 VJ=20.00
MOVJ C00106 BC00106 VJ=30.00  +MOVJ EC00106 VJ=30.00
MOVJ C00107 BC00107 VJ=100.00  +MOVJ EC00107 VJ=20.00
MOVJ C00108 BC00108 VJ=30.00  +MOVJ EC00108 VJ=30.00
SFTON3D P029
MOVJ C00109 BC00109 VJ=30.00  +MOVJ EC00109 VJ=30.00
SMOVL C00110 BC00110 V=166.7  +MOVJ EC00110
ARCON
SMOVL C00111 BC00111 V=10.0  +MOVJ EC00111
SFTOF3D
SFTON3D P030
SMOVL C00112 BC00112 V=10.0  +MOVJ EC00112
SMOVL C00113 BC00113 V=10.0  +MOVJ EC00113
SMOVL C00114 BC00114 V=10.0  +MOVJ EC00114
ARCOF
MOVJ C00115 BC00115 VJ=20.00  +MOVJ EC00115 VJ=20.00
SFTOF3D
MOVJ C00116 BC00116 VJ=100.00  +MOVJ EC00116 VJ=100.00
MOVJ C00117 BC00117 VJ=100.00  +MOVJ EC00117 VJ=100.00
SFTOF
CALL JOB:CLEAN-R1_KM_NEW_SCIANA
MOVJ C00118 BC00118 VJ=100.00  +MOVJ EC00118 VJ=100.00
'SZUKANIE DRUGA STRONA
MOVJ C00119 BC00119 VJ=30.00  +MOVJ EC00119 VJ=15.00
SFTOF3D
MOVL C00120 BC00120 V=83.3  +MOVJ EC00120 VJ=15.00
SREFP 3 C00121 BC00121  +REFP EC00121
CALL JOB:SEARCH-R1-S13D
SET P035 P006
SFTON3D P035
MOVL C00122 BC00122 V=83.3  +MOVJ EC00122 VJ=15.00
SREFP 3 C00123 BC00123  +REFP EC00123
CALL JOB:SEARCH-R1-S13D
SET P035 P006
MOVL C00124 BC00124 V=83.3  +MOVJ EC00124 VJ=15.00
SFTOF3D
MOVJ C00125 BC00125 VJ=50.00  +MOVJ EC00125 VJ=50.00
MOVJ C00126 BC00126 VJ=15.00  +MOVJ EC00126 VJ=15.00
MOVL C00127 BC00127 V=83.3  +MOVJ EC00127 VJ=15.00
MOVL C00128 BC00128 V=166.7  +MOVJ EC00128 VJ=15.00
SREFP 3 C00129 BC00129  +REFP EC00129
CALL JOB:SEARCH-R1-S13D
SET P026 P006
SFTON3D P026
MOVL C00130 BC00130 V=83.3  +MOVJ EC00130 VJ=15.00
SREFP 3 C00131 BC00131  +REFP EC00131
CALL JOB:SEARCH-R1-S13D
SET P026 P006
MOVL C00132 BC00132 V=83.3  +MOVJ EC00132 VJ=15.00
SFTOF3D
MOVL C00133 BC00133 V=250.0  +MOVJ EC00133 VJ=15.00
MOVL C00134 BC00134 V=166.7  +MOVJ EC00134 VJ=15.00
SREFP 3 C00135 BC00135  +REFP EC00135
CALL JOB:SEARCH-R1-S13D
SET P027 P006
SFTON3D P027
MOVL C00136 BC00136 V=250.0  +MOVJ EC00136 VJ=15.00
SREFP 3 C00137 BC00137  +REFP EC00137
CALL JOB:SEARCH-R1-S13D
SET P027 P006
MOVL C00138 BC00138 V=166.7  +MOVJ EC00138 VJ=15.00
SFTOF3D
SMOVL C00139 BC00139 V=250.0  +MOVJ EC00139
MOVL C00140 BC00140 V=250.0  +MOVJ EC00140 VJ=15.00
MOVL C00141 BC00141 V=250.0  +MOVJ EC00141 VJ=15.00
SREFP 3 C00142 BC00142  +REFP EC00142
CALL JOB:SEARCH-R1-S13D
SET P028 P006
SFTON3D P028
MOVL C00143 BC00143 V=83.3  +MOVJ EC00143 VJ=15.00
SREFP 3 C00144 BC00144  +REFP EC00144
CALL JOB:SEARCH-R1-S13D
SET P028 P006
MOVL C00145 BC00145 V=83.3  +MOVJ EC00145 VJ=15.00
SFTOF3D
MOVJ C00146 BC00146 VJ=15.00  +MOVJ EC00146 VJ=15.00
MOVJ C00147 BC00147 VJ=15.00  +MOVJ EC00147 VJ=15.00
SFTOF3D
MOVJ C00148 BC00148 VJ=15.00  +MOVJ EC00148 VJ=15.00
MOVL C00149 BC00149 V=83.3  +MOVJ EC00149 VJ=15.00
SREFP 3 C00150 BC00150  +REFP EC00150
CALL JOB:SEARCH-R1-S13D
SET P034 P006
SFTON3D P034
MOVL C00151 BC00151 V=83.3  +MOVJ EC00151 VJ=15.00
SREFP 3 C00152 BC00152  +REFP EC00152
CALL JOB:SEARCH-R1-S13D
SET P034 P006
MOVL C00153 BC00153 V=250.0  +MOVJ EC00153 VJ=15.00
MOVJ C00154 BC00154 VJ=15.00  +MOVJ EC00154 VJ=15.00
'KONIEC SZUKANIE DRUGA STRONA
'SPAWANIE DRUGA STRONA
MOVJ C00155 BC00155 VJ=15.00  +MOVJ EC00155 VJ=15.00
MACRO1 MJ#(0) ARGF7
SFTOF3D
SFTON3D P034
MOVJ C00156 BC00156 VJ=15.00  +MOVJ EC00156 VJ=15.00
SMOVL C00157 BC00157 V=250.0  +MOVJ EC00157
ARCON
SMOVL C00158 BC00158 V=10.0  +MOVJ EC00158
SFTOF3D
ARCOF
MOVJ C00159 BC00159 VJ=15.00  +MOVJ EC00159 VJ=15.00
MOVJ C00160 BC00160 VJ=50.00  +MOVJ EC00160 VJ=15.00
MOVJ C00161 BC00161 VJ=50.00  +MOVJ EC00161 VJ=50.00
MOVJ C00162 BC00162 VJ=50.00  +MOVJ EC00162 VJ=50.00
MOVJ C00163 BC00163 VJ=50.00  +MOVJ EC00163 VJ=50.00
SFTON3D P035
SMOVL C00164 BC00164 V=166.7  +MOVJ EC00164
ARCON
SMOVL C00165 BC00165 V=10.0  +MOVJ EC00165
SMOVL C00166 BC00166 V=10.0  +MOVJ EC00166
ARCOF
SFTOF3D
MOVJ C00167 BC00167 VJ=20.00  +MOVJ EC00167 VJ=50.00
MOVJ C00168 BC00168 VJ=50.00  +MOVJ EC00168 VJ=20.00
SFTON3D P027
MOVJ C00169 BC00169 VJ=20.00  +MOVJ EC00169 VJ=20.00
SMOVL C00170 BC00170 V=166.7  +MOVJ EC00170
ARCON
SMOVL C00171 BC00171 V=10.0  +MOVJ EC00171
SFTOF3D
SFTON3D P028
SMOVL C00172 BC00172 V=10.0  +MOVJ EC00172
ARCOF
MOVJ C00173 BC00173 VJ=20.00  +MOVJ EC00173 VJ=100.00
MOVJ C00174 BC00174 VJ=15.00  +MOVJ EC00174 VJ=15.00
SFTOF3D
MOVJ C00175 BC00175 VJ=15.00  +MOVJ EC00175 VJ=15.00
MOVJ C00176 BC00176 VJ=20.00  +MOVJ EC00176 VJ=20.00
SFTON3D P027
MOVJ C00177 BC00177 VJ=20.00  +MOVJ EC00177 VJ=20.00
SMOVL C00178 BC00178 V=10.0  +MOVJ EC00178
ARCON
SMOVL C00179 BC00179 V=10.0  +MOVJ EC00179
SFTOF3D
SFTON3D P026
SMOVL C00180 BC00180 V=10.0  +MOVJ EC00180
SMOVL C00181 BC00181 V=10.0  +MOVJ EC00181
ARCOF
MOVJ C00182 BC00182 VJ=15.00  +MOVJ EC00182 VJ=15.00
SFTOF3D
MOVJ C00183 BC00183 VJ=100.00  +MOVJ EC00183 VJ=15.00
MOVJ C00184 BC00184 VJ=100.00  +MOVJ EC00184 VJ=100.00
MOVJ C00185 BC00185 VJ=100.00  +MOVJ EC00185 VJ=100.00
MOVJ C00186 BC00186 VJ=100.00  +MOVJ EC00186 VJ=100.00
CALL JOB:CLEAN-R1_KM_NEW_SCIANA
MOVJ C00187 BC00187 VJ=100.00  +MOVJ EC00187 VJ=100.00
MOVJ C00188 BC00188 VJ=100.00  +MOVJ EC00188 VJ=100.00
MOVJ C00189 BC00189 VJ=100.00  +MOVJ EC00189 VJ=100.00
MOVL C00190 BC00190 V=166.7  +MOVJ EC00190 VJ=15.00
SREFP 3 C00191 BC00191  +REFP EC00191
CALL JOB:SEARCH-R1-S13D
SET P021 P006
SFTON3D P021
MOVL C00192 BC00192 V=83.3  +MOVJ EC00192 VJ=15.00
SREFP 3 C00193 BC00193  +REFP EC00193
CALL JOB:SEARCH-R1-S13D
SET P021 P006
MOVL C00194 BC00194 V=83.3  +MOVJ EC00194 VJ=15.00
SFTOF3D
MOVL C00195 BC00195 V=166.7  +MOVJ EC00195 VJ=15.00
MOVL C00196 BC00196 V=83.3  +MOVJ EC00196 VJ=15.00
SREFP 3 C00197 BC00197  +REFP EC00197
CALL JOB:SEARCH-R1-S13D
SET P022 P006
SFTON3D P022
MOVL C00198 BC00198 V=83.3  +MOVJ EC00198 VJ=15.00
REFP 3 RB1 C00199 BC00199
SREFP 3 C00200 BC00200  +REFP EC00199
CALL JOB:SEARCH-R1-S13D
SET P022 P006
MOVL C00201 BC00201 V=83.3  +MOVJ EC00200 VJ=15.00
SFTOF3D
MOVL C00202 BC00202 V=166.7  +MOVJ EC00201 VJ=15.00
MOVL C00203 BC00203 V=166.7  +MOVJ EC00202 VJ=15.00
SREFP 3 C00204 BC00204  +REFP EC00203
CALL JOB:SEARCH-R1-S13D
SET P023 P006
SFTON3D P023
MOVL C00205 BC00205 V=83.3  +MOVJ EC00204 VJ=15.00
SREFP 3 C00206 BC00206  +REFP EC00205
CALL JOB:SEARCH-R1-S13D
SET P023 P006
MOVL C00207 BC00207 V=83.3  +MOVJ EC00206 VJ=15.00
SFTOF3D
MOVL C00208 BC00208 V=166.7  +MOVJ EC00207 VJ=15.00
MOVL C00209 BC00209 V=166.7  +MOVJ EC00208 VJ=15.00
SREFP 3 C00210 BC00210  +REFP EC00209
CALL JOB:SEARCH-R1-S13D
SET P024 P006
SFTON3D P024
MOVL C00211 BC00211 V=83.3  +MOVJ EC00210 VJ=15.00
SREFP 3 C00212 BC00212  +REFP EC00211
CALL JOB:SEARCH-R1-S13D
SET P024 P006
MOVL C00213 BC00213 V=83.3  +MOVJ EC00212 VJ=15.00
SFTOF3D
MOVL C00214 BC00214 V=166.7  +MOVJ EC00213 VJ=15.00
MOVL C00215 BC00215 V=166.7  +MOVJ EC00214 VJ=15.00
SREFP 3 C00216 BC00216  +REFP EC00215
CALL JOB:SEARCH-R1-S13D
SET P025 P006
SFTON3D P025
MOVL C00217 BC00217 V=83.3  +MOVJ EC00216 VJ=15.00
SREFP 3 C00218 BC00218  +REFP EC00217
CALL JOB:SEARCH-R1-S13D
SET P025 P006
MOVL C00219 BC00219 V=133.3  +MOVJ EC00218 VJ=15.00
SFTOF3D
MOVJ C00220 BC00220 VJ=30.00  +MOVJ EC00219 VJ=100.00
MOVJ C00221 BC00221 VJ=30.00  +MOVJ EC00220 VJ=30.00
SFTON3D P023
MACRO1 MJ#(0) ARGF7
SMOVL C00222 BC00222 V=166.7  +MOVJ EC00221
ARCON
SFTOF3D
SFTON3D P022
SMOVL C00223 BC00223 V=10.8  +MOVJ EC00222
SFTOF3D
SFTON3D P021
SMOVL C00224 BC00224 V=10.8  +MOVJ EC00223
SMOVL C00225 BC00225 V=10.8  +MOVJ EC00224
ARCOF
SFTOF3D
MOVJ C00226 BC00226 VJ=30.00  +MOVJ EC00225 VJ=30.00
MOVJ C00227 BC00227 VJ=30.00  +MOVJ EC00226 VJ=30.00
SFTON3D P023
SMOVL C00228 BC00228 V=166.7  +MOVJ EC00227
ARCON
SFTOF3D
SFTON3D P024
SMOVL C00229 BC00229 V=10.8  +MOVJ EC00228
SFTOF3D
SFTON3D P025
SMOVL C00230 BC00230 V=10.8  +MOVJ EC00229
SMOVL C00231 BC00231 V=10.8  +MOVJ EC00230
SMOVL C00232 BC00232 V=10.8  +MOVJ EC00231
ARCOF
SFTOF3D
MOVJ C00233 BC00233 VJ=30.00  +MOVJ EC00232 VJ=30.00
MOVJ C00234 BC00234 VJ=30.00  +MOVJ EC00233 VJ=30.00
MOVJ C00235 BC00235 VJ=100.00  +MOVJ EC00234 VJ=100.00
MOVJ C00236 BC00236 VJ=30.00  +MOVJ EC00235 VJ=30.00
CALL JOB:ONLY_CUT_KM_NEW_SCIANA
MOVJ C00237 BC00237 VJ=30.00  +MOVJ EC00236 VJ=30.00
MOVJ C00238 BC00238 VJ=100.00  +MOVJ EC00237 VJ=100.00
MOVJ C00239 BC00239 VJ=60.00  +MOVJ EC00238 VJ=30.00
MOVJ C00240 BC00240 VJ=80.00  +MOVJ EC00239 VJ=80.00
MOVJ C00241 BC00241 VJ=20.00  +MOVJ EC00240 VJ=80.00
MOVJ C00242 BC00242 VJ=60.00  +MOVJ EC00241 VJ=30.00
MOVJ C00243 BC00243 VJ=60.00  +MOVJ EC00242 VJ=30.00
MOVJ C00244 BC00244 VJ=100.00  +MOVJ EC00243 VJ=100.00
MOVL C00245 BC00245 V=83.3  +MOVJ EC00244 VJ=15.00
SREFP 3 C00246 BC00246  +REFP EC00245
CALL JOB:SEARCH-R1-S13D
SET P021 P006
SFTON3D P021
MOVL C00247 BC00247 V=83.3  +MOVJ EC00246 VJ=15.00
SREFP 3 C00248 BC00248  +REFP EC00247
CALL JOB:SEARCH-R1-S13D
SET P021 P006
MOVL C00249 BC00249 V=83.3  +MOVJ EC00248 VJ=15.00
SFTOF3D
MOVL C00250 BC00250 V=166.7  +MOVJ EC00249 VJ=15.00
MOVL C00251 BC00251 V=83.3  +MOVJ EC00250 VJ=15.00
SREFP 3 C00252 BC00252  +REFP EC00251
CALL JOB:SEARCH-R1-S13D
SET P022 P006
SFTON3D P022
MOVL C00253 BC00253 V=83.3  +MOVJ EC00252 VJ=15.00
SREFP 3 C00254 BC00254  +REFP EC00253
CALL JOB:SEARCH-R1-S13D
SET P022 P006
MOVL C00255 BC00255 V=83.3  +MOVJ EC00254 VJ=15.00
SFTOF3D
MOVL C00256 BC00256 V=166.7  +MOVJ EC00255 VJ=15.00
MOVL C00257 BC00257 V=83.3  +MOVJ EC00256 VJ=15.00
SREFP 3 C00258 BC00258  +REFP EC00257
CALL JOB:SEARCH-R1-S13D
SET P023 P006
SFTON3D P023
MOVL C00259 BC00259 V=83.3  +MOVJ EC00258 VJ=15.00
SREFP 3 C00260 BC00260  +REFP EC00259
CALL JOB:SEARCH-R1-S13D
SET P023 P006
MOVL C00261 BC00261 V=83.3  +MOVJ EC00260 VJ=15.00
SFTOF3D
MOVL C00262 BC00262 V=166.7  +MOVJ EC00261 VJ=15.00
MOVL C00263 BC00263 V=166.7  +MOVJ EC00262 VJ=15.00
SREFP 3 C00264 BC00264  +REFP EC00263
CALL JOB:SEARCH-R1-S13D
SET P024 P006
SFTON3D P024
MOVL C00265 BC00265 V=83.3  +MOVJ EC00264 VJ=15.00
SREFP 3 C00266 BC00266  +REFP EC00265
CALL JOB:SEARCH-R1-S13D
SET P024 P006
MOVL C00267 BC00267 V=83.3  +MOVJ EC00266 VJ=15.00
SFTOF3D
MOVL C00268 BC00268 V=166.7  +MOVJ EC00267 VJ=15.00
MOVL C00269 BC00269 V=83.3  +MOVJ EC00268 VJ=15.00
SREFP 3 C00270 BC00270  +REFP EC00269
CALL JOB:SEARCH-R1-S13D
SET P025 P006
SFTON3D P025
MOVL C00271 BC00271 V=83.3  +MOVJ EC00270 VJ=15.00
SREFP 3 C00272 BC00272  +REFP EC00271
CALL JOB:SEARCH-R1-S13D
SET P025 P006
MOVL C00273 BC00273 V=166.7  +MOVJ EC00272 VJ=15.00
SFTOF3D
MOVJ C00274 BC00274 VJ=30.00  +MOVJ EC00273 VJ=100.00
MOVJ C00275 BC00275 VJ=30.00  +MOVJ EC00274 VJ=30.00
SFTON3D P023
MOVL C00276 BC00276 V=83.3  +MOVJ EC00275 VJ=30.00
ARCON
SFTOF3D
SFTON3D P022
MOVL C00277 BC00277 V=10.8  +MOVJ EC00276 VJ=30.00
SFTOF3D
SFTON3D P021
MOVL C00278 BC00278 V=10.8  +MOVJ EC00277 VJ=30.00
MOVL C00279 BC00279 V=10.8  +MOVJ EC00278 VJ=30.00
ARCOF
SFTOF3D
MOVJ C00280 BC00280 VJ=30.00  +MOVJ EC00279 VJ=30.00
MOVJ C00281 BC00281 VJ=30.00  +MOVJ EC00280 VJ=30.00
SFTON3D P023
MOVL C00282 BC00282 V=83.3  +MOVJ EC00281 VJ=30.00
ARCON
SFTOF3D
SFTON3D P024
MOVL C00283 BC00283 V=10.8  +MOVJ EC00282 VJ=30.00
SFTOF3D
SFTON3D P025
MOVL C00284 BC00284 V=10.8  +MOVJ EC00283 VJ=30.00
MOVL C00285 BC00285 V=10.8  +MOVJ EC00284 VJ=30.00
MOVL C00286 BC00286 V=10.8  +MOVJ EC00285 VJ=30.00
ARCOF
SFTOF3D
MOVJ C00287 BC00287 VJ=50.00  +MOVJ EC00286 VJ=30.00
MOVJ C00288 BC00288 VJ=50.00  +MOVJ EC00287 VJ=30.00
MOVJ C00289 BC00289 VJ=20.00  +MOVJ EC00288 VJ=20.00
MOVJ C00290 BC00290 VJ=50.00  +MOVJ EC00289 VJ=30.00
MOVJ C00291 BC00291 VJ=100.00  +MOVJ EC00290 VJ=100.00
PAUSE
PAUSE
'ZALOZYC USZY ZE SCIANY
MOVJ C00292 BC00292 VJ=100.00  +MOVJ EC00291 VJ=100.00
END
